(* Schneider Machine Expert - Basic project CONVEYOR_2_ZONE_ZPA_TM221CE24R, file version 3.0.0.0 *)
(* ProjectInformations: Name=New project *)

HARDWARE
  Cpu 0: TM221CE24R
  ModuleExtensionObject 0: TM3DI32K
  ModuleExtensionObject 1: TM3AI2H/G
  EthernetConfiguration: NetworkName=M221, IpAllocationMode=FixedAddress, IpAddress=0.0.0.0, SubnetMask=0.0.0.0
  SerialLineConfiguration: Baud=Baud19200, Parity=ParityEven, DataBits=DataBits8, StopBits=StopBits1, PhysicalMedium=PhysicalMediumRs485, TransmissionMode=TransmissionModeModbusRtu, SlaveId=1, Addressing=SlaveAddressing
  MastTask: UsePeriodScanMode=false, PeriodScan=100
  FastTask: Period=255
  CpuBehavior: StartingMode=StartAsPreviousState, AutoSaveRamOnEeprom=true, WatchdogPeriod=250

SYMBOLS  (address, symbol, comment, settings)
  %M0       AUTO_MODE  "1 = Auto; 0 = Manual"
  %M1       START_HMI  "Perintah Start HMI momentary"
  %M2       STOP_HMI  "Perintah Stop HMI"
  %M3       JOG_ZONE1  "Jog manual motor zona 1"
  %M4       JOG_ZONE2  "Jog manual motor zona 2"
  %M5       RESET_HMI  "Reset alarm dari HMI momentary"
  %M10      SYSTEM_RUN  "Latch sistem produksi"
  %M11      SAFETY_OK  "Ringkasan Stop E-Stop dan overload"
  %M12      AUTO_ZONE1_CMD  "Perintah otomatis zona 1"
  %M13      AUTO_ZONE2_CMD  "Perintah otomatis zona 2"
  %M14      FINAL_ZONE1_CMD  "Perintah akhir motor zona 1"
  %M15      FINAL_ZONE2_CMD  "Perintah akhir motor zona 2"
  %M20      JAM_ZONE1_LATCH  "Alarm macet zona 1 terlatch"
  %M21      JAM_ZONE2_LATCH  "Alarm macet zona 2 terlatch"
  %M22      ALARM_ACTIVE  "Alarm umum"
  %M23      RESET_REQUEST  "Gabungan reset panel dan HMI"
  %M30      PRODUCT_DEMAND_ZONE1  "Produk meminta zona 1 bergerak"
  %M31      MANUAL_JOG_ZONE1  "Perintah jog zona 1 tervalidasi"
  %M32      MANUAL_JOG_ZONE2  "Perintah jog zona 2 tervalidasi"
  %S6       SB_TB1S  "Time base of 1 s generated by an internal clock"
  %S13      SB_FIRSTRUN  "Indicates the first controller cycle in RUN mode"
  %MW1      WATER_RANGE_MM  "Range sensor level mm"
  %MW2      LEVEL_RAW_COPY  "Salinan raw input level"
  %MW10     MAX_HEIGHT_G1_MM  "Tinggi maksimum pintu 1 mm"
  %MW11     MAX_HEIGHT_G2_MM  "Tinggi maksimum pintu 2 mm"
  %MW12     MAX_HEIGHT_G3_MM  "Tinggi maksimum pintu 3 mm"
  %MW13     DEADBAND_PCT  "Deadband posisi persen"
  %MW20     ENC_ZERO_G1  "Nilai encoder pintu 1 saat tertutup"
  %MW21     ENC_ZERO_G2  "Nilai encoder pintu 2 saat tertutup"
  %MW22     ENC_ZERO_G3  "Nilai encoder pintu 3 saat tertutup"
  %MW23     ENC_SPAN_G1  "Span count tertutup-terbuka G1"
  %MW24     ENC_SPAN_G2  "Span count tertutup-terbuka G2"
  %MW25     ENC_SPAN_G3  "Span count tertutup-terbuka G3"
  %MW30     ENC_BINARY_G1  "Nilai biner encoder G1"
  %MW31     ENC_BINARY_G2  "Nilai biner encoder G2"
  %MW32     ENC_BINARY_G3  "Nilai biner encoder G3"
  %MW33     POS_COUNT_G1  "Count posisi terkoreksi G1"
  %MW34     POS_COUNT_G2  "Count posisi terkoreksi G2"
  %MW35     POS_COUNT_G3  "Count posisi terkoreksi G3"
  %MW50     TARGET_PCT_G1  "Target bukaan G1 0-100 persen"
  %MW51     TARGET_PCT_G2  "Target bukaan G2 0-100 persen"
  %MW52     TARGET_PCT_G3  "Target bukaan G3 0-100 persen"
  %MF60     POSITION_G1_PCT  "Posisi G1 persen"
  %MF62     POSITION_G2_PCT  "Posisi G2 persen"
  %MF64     POSITION_G3_PCT  "Posisi G3 persen"
  %MF66     POSITION_G1_MM  "Posisi G1 mm"
  %MF68     POSITION_G2_MM  "Posisi G2 mm"
  %MF70     POSITION_G3_MM  "Posisi G3 mm"
  %MF72     WATER_LEVEL_MM  "Level air mm"
  %MF74     WATER_LEVEL_PCT  "Level air persen"
  %MF76     WATER_RANGE_REAL  "Range level dalam REAL"
  %MF80     TARGET_G1_REAL  "Target G1 dalam REAL"
  %MF82     TARGET_G2_REAL  "Target G2 dalam REAL"
  %MF84     TARGET_G3_REAL  "Target G3 dalam REAL"
  %MF86     DEADBAND_REAL  "Deadband dalam REAL"
  %MF88     OPEN_THRESHOLD_G1  "Ambang buka G1"
  %MF90     CLOSE_THRESHOLD_G1  "Ambang tutup G1"
  %MF92     OPEN_THRESHOLD_G2  "Ambang buka G2"
  %MF94     CLOSE_THRESHOLD_G2  "Ambang tutup G2"
  %MF96     OPEN_THRESHOLD_G3  "Ambang buka G3"
  %MF98     CLOSE_THRESHOLD_G3  "Ambang tutup G3"
  %C0       JAM_SECONDS_ZONE1  "Counter pulsa 1 detik untuk jam zona 1; preset dinamis 8"
  %C1       JAM_SECONDS_ZONE2  "Counter pulsa 1 detik untuk jam zona 2; preset dinamis 8"
  %I0.0     START_PB  "Tombol Start NO"
  %I0.1     STOP_OK  "Kontak Stop NC; 1 = sehat"
  %I0.2     ESTOP_OK  "Feedback safety relay; 1 = sehat"
  %I0.3     OL_ZONE1_OK  "Kontak overload motor zona 1; 1 = sehat"
  %I0.4     OL_ZONE2_OK  "Kontak overload motor zona 2; 1 = sehat"
  %I0.5     SENSOR_INFEED  "Sensor produk masuk"
  %I0.6     SENSOR_ZONE1  "Sensor okupansi akhir zona 1"
  %I0.7     SENSOR_ZONE2  "Sensor okupansi akhir zona 2"
  %I0.8     DOWNSTREAM_READY  "Peralatan hilir siap menerima produk"
  %I0.9     RESET_PB  "Tombol reset alarm NO"
  %I0.10      "Tidak digunakan"
  %I0.11      "Tidak digunakan"
  %I0.12      "Tidak digunakan"
  %I0.13      "Tidak digunakan"
  %Q0.0     MOTOR_ZONE1  "Kontaktor atau VFD run motor zona 1"
  %Q0.1     MOTOR_ZONE2  "Kontaktor atau VFD run motor zona 2"
  %Q0.2       "Tidak digunakan"
  %Q0.3       "Tidak digunakan"
  %Q0.4     BUZZER  "Buzzer alarm umum"
  %Q0.5     LAMP_RUN  "Lampu sistem berjalan"
  %Q0.6     LAMP_FAULT  "Lampu fault"
  %Q0.7       "Tidak digunakan"
  %Q0.8       "Tidak digunakan"
  %Q0.9       "Tidak digunakan"
  %I1.0     ENC_G1_GRAY_B0  "E6CP pintu 1 Gray bit 0"
  %I1.1     ENC_G1_GRAY_B1  "E6CP pintu 1 Gray bit 1"
  %I1.2     ENC_G1_GRAY_B2  "E6CP pintu 1 Gray bit 2"
  %I1.3     ENC_G1_GRAY_B3  "E6CP pintu 1 Gray bit 3"
  %I1.4     ENC_G1_GRAY_B4  "E6CP pintu 1 Gray bit 4"
  %I1.5     ENC_G1_GRAY_B5  "E6CP pintu 1 Gray bit 5"
  %I1.6     ENC_G1_GRAY_B6  "E6CP pintu 1 Gray bit 6"
  %I1.7     ENC_G1_GRAY_B7  "E6CP pintu 1 Gray bit 7"
  %I1.8     ENC_G2_GRAY_B0  "E6CP pintu 2 Gray bit 0"
  %I1.9     ENC_G2_GRAY_B1  "E6CP pintu 2 Gray bit 1"
  %I1.10    ENC_G2_GRAY_B2  "E6CP pintu 2 Gray bit 2"
  %I1.11    ENC_G2_GRAY_B3  "E6CP pintu 2 Gray bit 3"
  %I1.12    ENC_G2_GRAY_B4  "E6CP pintu 2 Gray bit 4"
  %I1.13    ENC_G2_GRAY_B5  "E6CP pintu 2 Gray bit 5"
  %I1.14    ENC_G2_GRAY_B6  "E6CP pintu 2 Gray bit 6"
  %I1.15    ENC_G2_GRAY_B7  "E6CP pintu 2 Gray bit 7"
  %I1.16    ENC_G3_GRAY_B0  "E6CP pintu 3 Gray bit 0"
  %I1.17    ENC_G3_GRAY_B1  "E6CP pintu 3 Gray bit 1"
  %I1.18    ENC_G3_GRAY_B2  "E6CP pintu 3 Gray bit 2"
  %I1.19    ENC_G3_GRAY_B3  "E6CP pintu 3 Gray bit 3"
  %I1.20    ENC_G3_GRAY_B4  "E6CP pintu 3 Gray bit 4"
  %I1.21    ENC_G3_GRAY_B5  "E6CP pintu 3 Gray bit 5"
  %I1.22    ENC_G3_GRAY_B6  "E6CP pintu 3 Gray bit 6"
  %I1.23    ENC_G3_GRAY_B7  "E6CP pintu 3 Gray bit 7"
  %I1.24    MODE_AUTO  "Selector 1=AUTO 0=MANUAL"
  %I1.25    MAN_OPEN_G1  "PB manual buka pintu 1"
  %I1.26    MAN_CLOSE_G1  "PB manual tutup pintu 1"
  %I1.27    MAN_OPEN_G2  "PB manual buka pintu 2"
  %I1.28    MAN_CLOSE_G2  "PB manual tutup pintu 2"
  %I1.29    MAN_OPEN_G3  "PB manual buka pintu 3"
  %I1.30    MAN_CLOSE_G3  "PB manual tutup pintu 3"
  %I1.31    RESET_FAULT  "PB reset fault"
  %IW2.0    LEVEL_RAW  "Sensor level 4-20 mA raw 4000-20000"  [Type=Type_4_20mA, Scope=Scope_Customized, Minimum=4000, Maximum=20000]

POU CONVEYOR_2_ZONE_ZPA_IL
  (* SectionNumber=1 *)

// Rung 0: N01_SAFETY
// Ringkasan feedback Stop, E-Stop, overload, dan Stop HMI.
  LD %I0.1                (* STOP_OK *)
  AND %I0.2               (* ESTOP_OK *)
  AND %I0.3               (* OL_ZONE1_OK *)
  AND %I0.4               (* OL_ZONE2_OK *)
  ANDN %M2                (* STOP_HMI *)
  ST %M11                 (* SAFETY_OK *)
  // as ST:
  //   SAFETY_OK := STOP_OK AND ESTOP_OK AND OL_ZONE1_OK AND OL_ZONE2_OK AND NOT STOP_HMI;

// Rung 1: N02_RESET_REQUEST
// Gabungkan reset panel dan HMI.
  LD %I0.9                (* RESET_PB *)
  OR %M5                  (* RESET_HMI *)
  ST %M23                 (* RESET_REQUEST *)
  // as ST:
  //   RESET_REQUEST := RESET_PB OR RESET_HMI;

// Rung 2: N03_SYSTEM_RUN
// Latch produksi hanya pada mode Auto dan safety sehat.
  LD %I0.0                (* START_PB *)
  OR %M1                  (* START_HMI *)
  OR %M10                 (* SYSTEM_RUN *)
  AND %M0                 (* AUTO_MODE *)
  AND %M11                (* SAFETY_OK *)
  ST %M10                 (* SYSTEM_RUN *)
  // as ST:
  //   SYSTEM_RUN := (START_PB OR START_HMI OR SYSTEM_RUN) AND AUTO_MODE AND SAFETY_OK;

// Rung 3: N04_ZONE2_AUTO
// Zona 2 melepas produk hanya bila hilir siap.
  LD %M10                 (* SYSTEM_RUN *)
  AND %I0.7               (* SENSOR_ZONE2 *)
  AND %I0.8               (* DOWNSTREAM_READY *)
  ANDN %M22               (* ALARM_ACTIVE *)
  ST %M13                 (* AUTO_ZONE2_CMD *)
  // as ST:
  //   AUTO_ZONE2_CMD := SYSTEM_RUN AND SENSOR_ZONE2 AND DOWNSTREAM_READY AND NOT ALARM_ACTIVE;

// Rung 4: N05_ZONE1_DEMAND
// Produk masuk atau produk di ujung zona 1 menjadi demand.
  LD %I0.5                (* SENSOR_INFEED *)
  OR %I0.6                (* SENSOR_ZONE1 *)
  ST %M30                 (* PRODUCT_DEMAND_ZONE1 *)
  // as ST:
  //   PRODUCT_DEMAND_ZONE1 := SENSOR_INFEED OR SENSOR_ZONE1;

// Rung 5: N06_ZONE1_AUTO
// Zona 1 bergerak bila zona 2 kosong atau sedang melepas.
  LDN %I0.7               (* SENSOR_ZONE2 *)
  OR %M13                 (* AUTO_ZONE2_CMD *)
  AND %M10                (* SYSTEM_RUN *)
  ANDN %M22               (* ALARM_ACTIVE *)
  AND %M30                (* PRODUCT_DEMAND_ZONE1 *)
  ST %M12                 (* AUTO_ZONE1_CMD *)
  // as ST:
  //   AUTO_ZONE1_CMD := (NOT SENSOR_ZONE2 OR AUTO_ZONE2_CMD) AND SYSTEM_RUN AND NOT ALARM_ACTIVE AND PRODUCT_DEMAND_ZONE1;

// Rung 6: N07_JOG_ZONE1
// Validasi jog zona 1 hanya pada mode Manual.
  LD %M3                  (* JOG_ZONE1 *)
  ANDN %M0                (* AUTO_MODE *)
  ST %M31                 (* MANUAL_JOG_ZONE1 *)
  // as ST:
  //   MANUAL_JOG_ZONE1 := JOG_ZONE1 AND NOT AUTO_MODE;

// Rung 7: N08_JOG_ZONE2
// Validasi jog zona 2 hanya pada mode Manual.
  LD %M4                  (* JOG_ZONE2 *)
  ANDN %M0                (* AUTO_MODE *)
  ST %M32                 (* MANUAL_JOG_ZONE2 *)
  // as ST:
  //   MANUAL_JOG_ZONE2 := JOG_ZONE2 AND NOT AUTO_MODE;

// Rung 8: N09_FINAL_ZONE1
// Gabungkan Auto/Jog dengan interlock.
  LD %M12                 (* AUTO_ZONE1_CMD *)
  OR %M31                 (* MANUAL_JOG_ZONE1 *)
  AND %M11                (* SAFETY_OK *)
  ANDN %M22               (* ALARM_ACTIVE *)
  ST %M14                 (* FINAL_ZONE1_CMD *)
  // as ST:
  //   FINAL_ZONE1_CMD := (AUTO_ZONE1_CMD OR MANUAL_JOG_ZONE1) AND SAFETY_OK AND NOT ALARM_ACTIVE;

// Rung 9: N10_FINAL_ZONE2
// Gabungkan Auto/Jog dengan interlock.
  LD %M13                 (* AUTO_ZONE2_CMD *)
  OR %M32                 (* MANUAL_JOG_ZONE2 *)
  AND %M11                (* SAFETY_OK *)
  ANDN %M22               (* ALARM_ACTIVE *)
  ST %M15                 (* FINAL_ZONE2_CMD *)
  // as ST:
  //   FINAL_ZONE2_CMD := (AUTO_ZONE2_CMD OR MANUAL_JOG_ZONE2) AND SAFETY_OK AND NOT ALARM_ACTIVE;

// Rung 10: N11_COUNTER_PRESET_Z1
// Preset jam zona 1 = 8 pulsa; gunakan operation block M221.
  LD %S13                 (* SB_FIRSTRUN *)
  [ %C0.P := 8 ]          (* JAM_SECONDS_ZONE1 *)
  // as ST:
  //   IF SB_FIRSTRUN THEN JAM_SECONDS_ZONE1.P := 8; END_IF;

// Rung 11: N12_JAM_COUNTER_Z1
// Hitung tepi naik pulsa sistem saat motor diperintah dan sensor zona 1 tetap tertutup.
  BLK %C0                 (* JAM_SECONDS_ZONE1 *)
  LD %S6                  (* SB_TB1S *)
  AND %M14                (* FINAL_ZONE1_CMD *)
  AND %I0.6               (* SENSOR_ZONE1 *)
  CU
  LDN %M14                (* FINAL_ZONE1_CMD *)
  ORN %I0.6               (* SENSOR_ZONE1 *)
  R
  END_BLK
  // as ST:
  //   JAM_SECONDS_ZONE1(CU := SB_TB1S AND FINAL_ZONE1_CMD AND SENSOR_ZONE1, R := NOT FINAL_ZONE1_CMD OR NOT SENSOR_ZONE1);

// Rung 12: N13_COUNTER_PRESET_Z2
// Preset jam zona 2 = 8 pulsa; gunakan operation block M221.
  LD %S13                 (* SB_FIRSTRUN *)
  [ %C1.P := 8 ]          (* JAM_SECONDS_ZONE2 *)
  // as ST:
  //   IF SB_FIRSTRUN THEN JAM_SECONDS_ZONE2.P := 8; END_IF;

// Rung 13: N14_JAM_COUNTER_Z2
// Hitung tepi naik pulsa sistem saat motor diperintah dan sensor zona 2 tetap tertutup.
  BLK %C1                 (* JAM_SECONDS_ZONE2 *)
  LD %S6                  (* SB_TB1S *)
  AND %M15                (* FINAL_ZONE2_CMD *)
  AND %I0.7               (* SENSOR_ZONE2 *)
  CU
  LDN %M15                (* FINAL_ZONE2_CMD *)
  ORN %I0.7               (* SENSOR_ZONE2 *)
  R
  END_BLK
  // as ST:
  //   JAM_SECONDS_ZONE2(CU := SB_TB1S AND FINAL_ZONE2_CMD AND SENSOR_ZONE2, R := NOT FINAL_ZONE2_CMD OR NOT SENSOR_ZONE2);

// Rung 14: N15_LATCH_JAM_Z1
// Latch alarm saat counter zona 1 selesai.
  LD %C0.D                (* JAM_SECONDS_ZONE1 *)
  S %M20                  (* JAM_ZONE1_LATCH *)
  // as ST:
  //   IF JAM_SECONDS_ZONE1.D THEN JAM_ZONE1_LATCH := TRUE; END_IF;

// Rung 15: N16_LATCH_JAM_Z2
// Latch alarm saat counter zona 2 selesai.
  LD %C1.D                (* JAM_SECONDS_ZONE2 *)
  S %M21                  (* JAM_ZONE2_LATCH *)
  // as ST:
  //   IF JAM_SECONDS_ZONE2.D THEN JAM_ZONE2_LATCH := TRUE; END_IF;

// Rung 16: N17_RESET_JAM_Z1
// Reset zona 1 hanya bila sensor sudah bebas.
  LD %M23                 (* RESET_REQUEST *)
  ANDN %I0.6              (* SENSOR_ZONE1 *)
  R %M20                  (* JAM_ZONE1_LATCH *)
  // as ST:
  //   IF RESET_REQUEST AND NOT SENSOR_ZONE1 THEN JAM_ZONE1_LATCH := FALSE; END_IF;

// Rung 17: N18_RESET_JAM_Z2
// Reset zona 2 hanya bila sensor sudah bebas.
  LD %M23                 (* RESET_REQUEST *)
  ANDN %I0.7              (* SENSOR_ZONE2 *)
  R %M21                  (* JAM_ZONE2_LATCH *)
  // as ST:
  //   IF RESET_REQUEST AND NOT SENSOR_ZONE2 THEN JAM_ZONE2_LATCH := FALSE; END_IF;

// Rung 18: N19_ALARM_SUMMARY
// Alarm jam, E-Stop, atau overload.
  LD %M20                 (* JAM_ZONE1_LATCH *)
  OR %M21                 (* JAM_ZONE2_LATCH *)
  ORN %I0.2               (* ESTOP_OK *)
  ORN %I0.3               (* OL_ZONE1_OK *)
  ORN %I0.4               (* OL_ZONE2_OK *)
  ST %M22                 (* ALARM_ACTIVE *)
  // as ST:
  //   ALARM_ACTIVE := JAM_ZONE1_LATCH OR JAM_ZONE2_LATCH OR NOT ESTOP_OK OR NOT OL_ZONE1_OK OR NOT OL_ZONE2_OK;

// Rung 19: N20_OUTPUT_ZONE1
// Output fisik motor zona 1.
  LD %M14                 (* FINAL_ZONE1_CMD *)
  ST %Q0.0                (* MOTOR_ZONE1 *)
  // as ST:
  //   MOTOR_ZONE1 := FINAL_ZONE1_CMD;

// Rung 20: N21_OUTPUT_ZONE2
// Output fisik motor zona 2.
  LD %M15                 (* FINAL_ZONE2_CMD *)
  ST %Q0.1                (* MOTOR_ZONE2 *)
  // as ST:
  //   MOTOR_ZONE2 := FINAL_ZONE2_CMD;

// Rung 21: N22_LAMP_RUN
// Lampu Run aktif saat produksi Auto sehat.
  LD %M10                 (* SYSTEM_RUN *)
  ANDN %M22               (* ALARM_ACTIVE *)
  ST %Q0.5                (* LAMP_RUN *)
  // as ST:
  //   LAMP_RUN := SYSTEM_RUN AND NOT ALARM_ACTIVE;

// Rung 22: N23_FAULT_OUTPUTS
// Lampu fault dan buzzer mengikuti alarm umum.
  LD %M22                 (* ALARM_ACTIVE *)
  ST %Q0.6                (* LAMP_FAULT *)
  ST %Q0.4                (* BUZZER *)
  // as ST:
  //   LAMP_FAULT := ALARM_ACTIVE;
  //   BUZZER := ALARM_ACTIVE;
